PROGRAM ST5_MOTOR
VAR
	ClearFault: FB_ClearFault;
	SetEnableState: FB_SetEnableState;
	SetHomingParameter: FB_SetHomingParameter;
	FindHome: FB_FindHome;
	POSITION: DINT;
	GetMovementState: FB_GetMovementState;
	MoveToPosition: FB_MoveToPosition;
	SetOperationMode: FB_SetOperationMode;
	SetMotorParameter: FB_SetMotorParameter;
	SetPositionProfile: FB_SetPositionProfile;
END_VAR

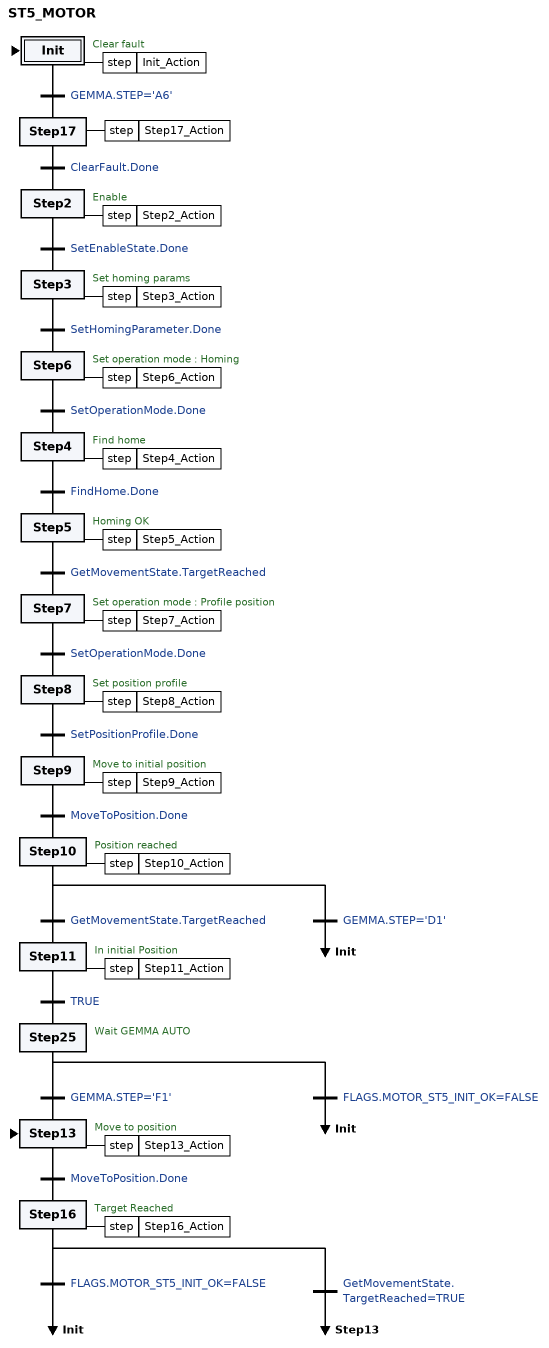
// Clear fault
INITIAL_STEP Init:
    Init_Action(N);  // step action
END_STEP
TRANSITION FROM Init TO Step17
    := GEMMA.STEP='A6';
END_TRANSITION
STEP Step17:
    Step17_Action(N);  // step action
END_STEP
TRANSITION FROM Step17 TO Step2
    := ClearFault.Done;
END_TRANSITION
// Enable
STEP Step2:
    Step2_Action(N);  // step action
END_STEP
TRANSITION FROM Step2 TO Step3
    := SetEnableState.Done;
END_TRANSITION
// Set homing params
STEP Step3:
    Step3_Action(N);  // step action
END_STEP
TRANSITION FROM Step3 TO Step6
    := SetHomingParameter.Done;
END_TRANSITION
// Set operation mode : Homing
STEP Step6:
    Step6_Action(N);  // step action
END_STEP
TRANSITION FROM Step6 TO Step4
    := SetOperationMode.Done;
END_TRANSITION
// Find home
STEP Step4:
    Step4_Action(N);  // step action
END_STEP
TRANSITION FROM Step4 TO Step5
    := FindHome.Done;
END_TRANSITION
// Homing OK
STEP Step5:
    Step5_Action(N);  // step action
END_STEP
TRANSITION FROM Step5 TO Step7
    := GetMovementState.TargetReached;
END_TRANSITION
// Set operation mode : Profile position
STEP Step7:
    Step7_Action(N);  // step action
END_STEP
TRANSITION FROM Step7 TO Step8
    := SetOperationMode.Done;
END_TRANSITION
// Set position profile
STEP Step8:
    Step8_Action(N);  // step action
END_STEP
TRANSITION FROM Step8 TO Step9
    := SetPositionProfile.Done;
END_TRANSITION
// Move to initial position
STEP Step9:
    Step9_Action(N);  // step action
END_STEP
TRANSITION FROM Step9 TO Step10
    := MoveToPosition.Done;
END_TRANSITION
// Position reached
STEP Step10:
    Step10_Action(N);  // step action
END_STEP
TRANSITION FROM Step10 TO Step11
    := GetMovementState.TargetReached;
END_TRANSITION
TRANSITION FROM Step10 TO Init
    := GEMMA.STEP='D1';
END_TRANSITION
// In initial Position
STEP Step11:
    Step11_Action(N);  // step action
END_STEP
TRANSITION FROM Step11 TO Step25
    := TRUE;
END_TRANSITION
// Wait GEMMA AUTO
STEP Step25:
END_STEP
TRANSITION FROM Step25 TO Step13
    := GEMMA.STEP='F1';
END_TRANSITION
TRANSITION FROM Step25 TO Init
    := FLAGS.MOTOR_ST5_INIT_OK=FALSE;
END_TRANSITION
// Move to position
STEP Step13:
    Step13_Action(N);  // step action
END_STEP
TRANSITION FROM Step13 TO Step16
    := MoveToPosition.Done;
END_TRANSITION
// Target Reached
STEP Step16:
    Step16_Action(N);  // step action
END_STEP
TRANSITION FROM Step16 TO Init
    := FLAGS.MOTOR_ST5_INIT_OK=FALSE;
END_TRANSITION
TRANSITION FROM Step16 TO Step13
    := GetMovementState.TargetReached=TRUE;
END_TRANSITION

ACTION Step2_Action:
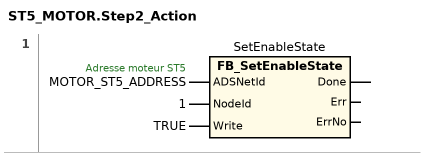
// NETWORK 1
//   MOTOR_ST5_ADDRESS: Adresse moteur ST5
SetEnableState(ADSNetId := MOTOR_ST5_ADDRESS, NodeId := 1, Write := TRUE); // FB_SetEnableState
END_ACTION

ACTION Step16_Action:
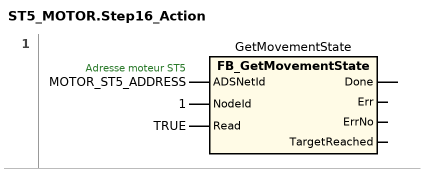
// NETWORK 1
//   MOTOR_ST5_ADDRESS: Adresse moteur ST5
GetMovementState(ADSNetId := MOTOR_ST5_ADDRESS, NodeId := 1, Read := TRUE); // FB_GetMovementState
END_ACTION

ACTION Step13_Action:
(*Limitation deplacement Moteur*)
IF FLAGS.MOTOR_ST5_POSITION>MOTOR_ST5_POSITION_MAX THEN
	POSITION:=MOTOR_ST5_POSITION_MAX;
ELSIF FLAGS.MOTOR_ST5_POSITION<0 THEN
	POSITION:=0;
ELSE
	POSITION:=FLAGS.MOTOR_ST5_POSITION;
END_IF


MoveToPosition(
	ADSNetId:= MOTOR_ST5_ADDRESS,
	NodeId:= 1,
	Write:= TRUE,
	TargetPosition:= POSITION,
	Absolut:= TRUE);
END_ACTION

ACTION Step5_Action:
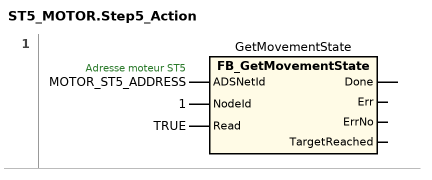
// NETWORK 1
//   MOTOR_ST5_ADDRESS: Adresse moteur ST5
GetMovementState(ADSNetId := MOTOR_ST5_ADDRESS, NodeId := 1, Read := TRUE); // FB_GetMovementState
END_ACTION

ACTION Step10_Action:
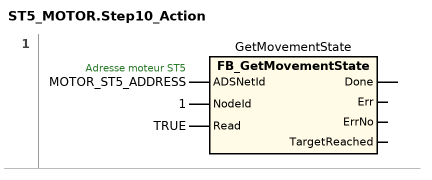
// NETWORK 1
//   MOTOR_ST5_ADDRESS: Adresse moteur ST5
GetMovementState(ADSNetId := MOTOR_ST5_ADDRESS, NodeId := 1, Read := TRUE); // FB_GetMovementState
END_ACTION

ACTION Step9_Action:
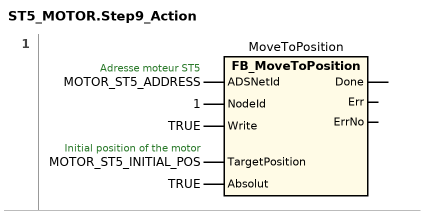
// NETWORK 1
//   MOTOR_ST5_ADDRESS: Adresse moteur ST5
//   MOTOR_ST5_INITIAL_POS: Initial position of the motor
MoveToPosition(
    ADSNetId := MOTOR_ST5_ADDRESS,
    NodeId := 1,
    Write := TRUE,
    TargetPosition := MOTOR_ST5_INITIAL_POS,
    Absolut := TRUE); // FB_MoveToPosition
END_ACTION

ACTION Step11_Action:

(*SetDisableState(
	ADSNetId:= '10.0.0.31.6.1',
	NodeId:= 1,
	Write:= TRUE);*)

FLAGS.MOTOR_ST5_INIT_OK:=TRUE;
END_ACTION

ACTION Step8_Action:
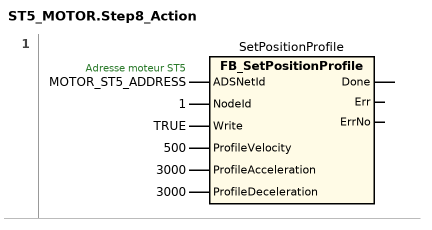
// NETWORK 1
//   MOTOR_ST5_ADDRESS: Adresse moteur ST5
SetPositionProfile(
    ADSNetId := MOTOR_ST5_ADDRESS,
    NodeId := 1,
    Write := TRUE,
    ProfileVelocity := 500,
    ProfileAcceleration := 3000,
    ProfileDeceleration := 3000); // FB_SetPositionProfile
END_ACTION

ACTION Step6_Action:
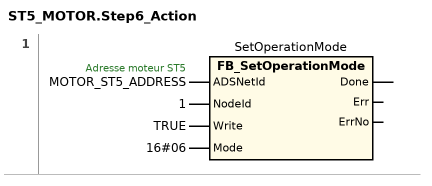
// NETWORK 1
//   MOTOR_ST5_ADDRESS: Adresse moteur ST5
SetOperationMode(ADSNetId := MOTOR_ST5_ADDRESS, NodeId := 1, Write := TRUE, Mode := 16#06); // FB_SetOperationMode
END_ACTION

ACTION Init_Action:

END_ACTION

ACTION Step3_Action:
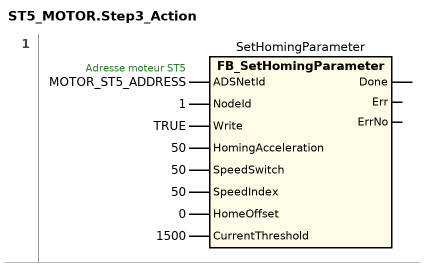
// NETWORK 1
//   MOTOR_ST5_ADDRESS: Adresse moteur ST5
SetHomingParameter(
    ADSNetId := MOTOR_ST5_ADDRESS,
    NodeId := 1,
    Write := TRUE,
    HomingAcceleration := 50,
    SpeedSwitch := 50,
    SpeedIndex := 50,
    HomeOffset := 0,
    CurrentThreshold := 1500); // FB_SetHomingParameter
END_ACTION

ACTION Step17_Action:
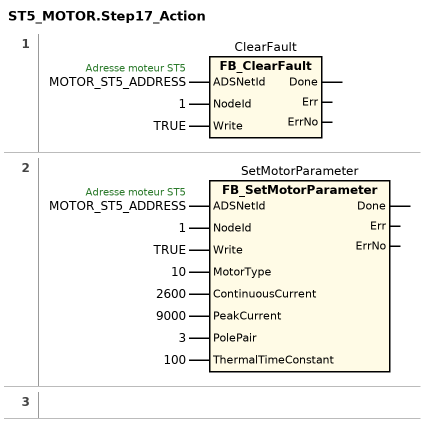
// NETWORK 1
//   MOTOR_ST5_ADDRESS: Adresse moteur ST5
ClearFault(ADSNetId := MOTOR_ST5_ADDRESS, NodeId := 1, Write := TRUE); // FB_ClearFault

// NETWORK 2
//   MOTOR_ST5_ADDRESS: Adresse moteur ST5
SetMotorParameter(
    ADSNetId := MOTOR_ST5_ADDRESS,
    NodeId := 1,
    Write := TRUE,
    MotorType := 10,
    ContinuousCurrent := 2600,
    PeakCurrent := 9000,
    PolePair := 3,
    ThermalTimeConstant := 100); // FB_SetMotorParameter

// NETWORK 3
END_ACTION

ACTION Step4_Action:
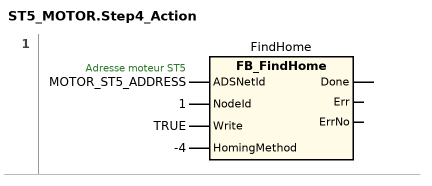
// NETWORK 1
//   MOTOR_ST5_ADDRESS: Adresse moteur ST5
FindHome(ADSNetId := MOTOR_ST5_ADDRESS, NodeId := 1, Write := TRUE, HomingMethod := -4); // FB_FindHome
END_ACTION

ACTION Step7_Action:
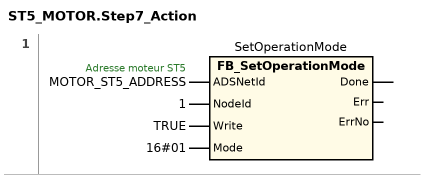
// NETWORK 1
//   MOTOR_ST5_ADDRESS: Adresse moteur ST5
SetOperationMode(ADSNetId := MOTOR_ST5_ADDRESS, NodeId := 1, Write := TRUE, Mode := 16#01); // FB_SetOperationMode
END_ACTION

END_PROGRAM

(* stored: Version 1.1.0.1, ProductVersion 3.1.0.26
   POU ST5_MOTOR: Id {eaa22ce4-e2ab-4cbd-b43f-2fea7879107c}
   Action Step2_Action: Id {17a1f33c-3aee-4969-91c1-e2232252da84}
   Action Step16_Action: Id {2de5a297-009e-46a4-bd7e-8f37de04ded6}
   Action Step13_Action: Id {35fcf7ba-92d5-4619-9995-0d37781c6798}
   Action Step5_Action: Id {4f097aee-3e1c-4eca-9fc9-0900ef97f55a}
   Action Step10_Action: Id {567083d5-13e2-4361-a749-33e108f4c5a0}
   Action Step9_Action: Id {5fdd8910-1b74-4874-8e0e-7ed6049c09b0}
   Action Step11_Action: Id {81cc9efc-8fac-431e-91f4-1247599f7540}
   Action Step8_Action: Id {b9bc49a8-9d6b-43ad-834a-b73ed28669ea}
   Action Step6_Action: Id {c278766a-4a92-4495-a124-553c3e7f4907}
   Action Init_Action: Id {c672e744-dc4a-4f7b-b2de-023d62f7658a}
   Action Step3_Action: Id {d4f76e97-91bf-40a1-badd-1667e87b929a}
   Action Step17_Action: Id {edf5214e-c385-44a3-a6b6-051088638e80}
   Action Step4_Action: Id {f8896a3d-408c-4ec0-832f-95425c85fd84}
   Action Step7_Action: Id {fc3e7d78-3fd8-46e6-ada8-fc5cb80a21d8} *)
